PROGRAM PRG_Kitchen
VAR
	fbLamp : ARRAY[0..1] OF FB_Lamp;
	fbDimmer : ARRAY[0..1] OF FB_Dimmer;
	i: INT;	
END_VAR


	FOR i := 0 TO 1 BY 1 DO
		fbLamp[i]();
		fbDimmer[i]();
	END_FOR

END_PROGRAM

(* stored: Version 1.1.0.1, ProductVersion 3.1.4024.12
   POU PRG_Kitchen: Id {6b282e00-63f8-43ea-bd6b-6706bbeae6e4}, SpecialFunc None *)
